(* IEC 61131-3 sources: lc3-arduino-ethernet/src/movinglight, 3 files *)

(* ---- ControllinoIoAccess.iecst ---- *)
/*
 * This function initializes required IO lines
 */
FUNCTION ControllinoInitialize
	VAR
		cnt : USINT;
	END_VAR
	FOR cnt := 0 TO GetNumberOfLEDs() DO
		ArduinoPinMode(pin := ControllinoMapDigitalOutputIdxToPin(cnt), mode := ArduinoPinDirection#OUTPUT);
	END_FOR;
	FOR cnt := 0 TO GetNumberOfInputs() DO
		ArduinoPinMode(pin := ControllinoMapDigitalInputIdxToPin(cnt), mode := ArduinoPinDirection#INPUT);
	END_FOR;
END_FUNCTION

/*
 * This function transfers data from Controllino inputs to global variables used in the logic
 */
FUNCTION MapInputsToVariables
	VAR_EXTERNAL
		switchInvert : BOOL;
	END_VAR
	VAR
		pinInput : USINT;
	END_VAR

	pinInput := ControllinoMapDigitalInputIdxToPin(index := 0, ENO => ENO);
	IF NOT ENO THEN
		RETURN;
	END_IF;
	switchInvert := ArduinoDigitalRead(pin := pinInput);
END_FUNCTION

/*
 * This function transfers data from the global variables used in the logic to the Controllino outputs
 */
FUNCTION MapVariablesToOutputs
	VAR_EXTERNAL
		outLedPattern     : LWORD;
	END_VAR
	VAR
		cnt : USINT;
	END_VAR

	FOR cnt := 0 TO GetNumberOfLEDs() DO
		ArduinoDigitalWrite(pin := ControllinoMapDigitalOutputIdxToPin(cnt), value := BIT_TST(outLedPattern,cnt));
	END_FOR;
END_FUNCTION

(* ---- MovingLight.iecst ---- *)
/*
 * This is an example for controlling and shifting LEDs of the hardware, when activating a push button on the hardware:
 *   If the push button on the hardware is pressed down, the LEDs are inverted.
 */
FUNCTION_BLOCK MovingLight
	VAR_INPUT
	/* different platforms have a different number of LEDs */
		numberOfLEDs : USINT;
	END_VAR
	VAR
		data : MovingLight_Data;

		SetModesAccordingToInputs : MovingLight_SetModesAccordingToInputs;
	END_VAR

	/* At least one LED must be turned on */
	IF data.ledPattern = 0 THEN
		data.ledPattern := 16#08;
	END_IF;

	SetModesAccordingToInputs(data := data);
	MovingLight_ShiftPatternAccordingToShiftDirection(data := data);
	MovingLight_HandleDirectionChange(numberOfLeftMostLED := numberOfLEDs - 1, data := data);
	MovingLight_WritePatternToOutput(data := data);

END_FUNCTION_BLOCK

/*
 * instance data for moving light module
 */
TYPE
	MovingLight_Data : STRUCT
	/* shift direction (true = shift left, false = shift right */
		shiftLeft : BOOL;
		/* invert pattern */
		invertLeds : BOOL;
		/* internal led pattern */
		ledPattern : LWORD;
	END_STRUCT;
END_TYPE

/*
 * changes modes if rising edge of input is detected:
 *   switchInvert: toggle invert mode
 */
FUNCTION_BLOCK MovingLight_SetModesAccordingToInputs
	VAR_IN_OUT
		data : MovingLight_Data;
	END_VAR

	VAR
		invertTrigger : R_TRIG;
	END_VAR

	VAR_EXTERNAL
		switchInvert : BOOL;
	END_VAR

	/* If the push button is pressed down, invert mode is toggled */
	IF invertTrigger.Q THEN
		data.invertLeds := NOT data.invertLeds;
	END_IF;

END_FUNCTION_BLOCK

/*
 * in cycle mode, changes shift direction if left/rightmost led is on
 */
FUNCTION MovingLight_HandleDirectionChange
	VAR_INPUT
	/* different platforms have a different number of LEDs */
		numberOfLeftMostLED : USINT;
	END_VAR

	VAR_IN_OUT
		data : MovingLight_Data;
	END_VAR

	/* set direction to right if leftmost led is on */
	IF BIT_TST(IN := data.ledPattern, N := numberOfLeftMostLED) THEN
		data.shiftLeft := FALSE;
		/* set direction to left if rightmost led is on */
	ELSIF BIT_TST(IN := data.ledPattern, N := 0) THEN
		data.shiftLeft := TRUE;
	END_IF;

END_FUNCTION

FUNCTION MovingLight_ShiftPatternAccordingToShiftDirection
	VAR_IN_OUT
		data : MovingLight_Data;
	END_VAR

	IF data.shiftLeft THEN
		/* Rotate the LEDs to the left */
		data.ledPattern := ROL(IN := data.ledPattern, N := 1);
	ELSE
	/* Rotate the LEDs to the right */
		data.ledPattern := ROR(IN := data.ledPattern, N := 1);
	END_IF;

END_FUNCTION

FUNCTION MovingLight_WritePatternToOutput
	VAR_IN_OUT
		data : MovingLight_Data;
	END_VAR

	VAR_EXTERNAL
		outLedPattern : LWORD;
	END_VAR

	IF data.invertLeds THEN
		outLedPattern := NOT data.ledPattern;
	ELSE
		outLedPattern := data.ledPattern;
	END_IF;

END_FUNCTION

(* ---- program_local.iecst ---- *)
/*
 * This is the main program for the simulation of the moving light example for the local plc.  <br/>
 * Only the program logic is executed.                                                         <br/>
 */
PROGRAM MovingLightSimulation
	VAR_GLOBAL
		switchInvert : BOOL;
		outLedPattern : LWORD;
	END_VAR

	VAR
		movingLight : MovingLight;
		stringPattern : STRING[64];
	END_VAR

	movingLight(numberOfLEDs:=GetNumberOfLEDs());

	stringPattern := PrepareString(outLedPattern);

END_PROGRAM

FUNCTION PrepareString : STRING[64]
      VAR_INPUT
            pattern : LWORD;
      END_VAR
      VAR
            idx : USINT;
      END_VAR

      FOR idx := 0 TO 63 DO
        if (BIT_TST(pattern, 63 - idx)) THEN
            PrepareString[idx] := 'X';
        ELSE
            PrepareString[idx] := '-';
        END_IF;
      END_FOR;
END_FUNCTION
